(* Logix 5000 project; controller Receptivo vendor 1 type 14 code 106 rev 30.11; software revision 30.00; part 5 of 10 *)
(* tags used below, declared in another part *)
   Codigo_QAD1_Espacios : DINT;
   Descripcion1_Espacios : DINT;
   Descripcion2_Espacios : DINT;
   Numero_Espacios_Descripcion_1 : DINT;
   Numero_Espacios_Descripcion_2 : DINT;
   Numero_Espacios_QAD1 : DINT;
   Numero_Espacios_QAD2 : DINT;
   Print1_Ejecute : BOOL;
   Print1_OK : BOOL;
   Print2_Ejecute : BOOL;
   Print2_OK : BOOL;
   CAJAS_1 : DINT;
   CAJAS_2 : DINT;
   Calendario : Hora_y_Fecha;
   Cant_total : SINT;
   CERO : DINT;
   Clima_1 : DINT;
   Clima_2 : DINT;
   Codigo_QAD2_Espacios : DINT;
   Consecutivo : INT;
   Consecutivo_String : Consecutivo;
   Consolidado_Est : UDT_COLA[50];
   Counter_R_Estacion1 : COUNTER;
   Counter_R_Estacion2 : COUNTER;
   Counter_R_Estacion3 : COUNTER;
   Counter_R_Estacion4 : COUNTER;
   Densidad_1 : REAL;
   Densidad_2 : REAL;
   Densidad_Elmar_1 : REAL;
   Densidad_Fogg1_1 : REAL;
   EAN14_1 : Codigo_Barras;
   EAN14_2 : Codigo_Barras;
   Espacios : STRING;
   ESTACION_1 : DINT;
   Estacion_1_GCola_1 : UDT_COLA;
   Estacion_1_General : UDT_GENERAL;
   Estacion_1_Resumen : UDT_COLA[20];
   Estacion_1_String : STRING;
   ESTACION_2 : DINT;
   Estacion_2_GCola_1 : UDT_COLA;
   Estacion_2_General : UDT_GENERAL;
   Estacion_2_Resumen : UDT_COLA[20];
   Estacion_2_String : STRING;
   Estacion_3_Resumen : UDT_COLA[20];
   Estacion_4_Resumen : UDT_COLA[20];
   Forx : SINT;
   Fory : SINT;
   Forz : SINT;
   found : SINT;
   LInea_General_1 : INT;
   LInea_General_2 : INT;
   Linea_String_General : STRING;
   Lote : DINT;
   Operador_1 : DINT;
   Operador_2 : DINT;
   Pesaje_1 : REAL;
   Pesaje_2 : REAL;
   Peso_Caja_Elmar_1 : REAL;
   Peso_Caja_Fogg1_1 : REAL;
   PESO_REAL_1 : DINT;
   PESO_REAL_2 : DINT;
   PESO_TEORICO_1 : DINT;
   PESO_TEORICO_2 : DINT;
   Producido_Elmar_Ahora : UDT_Maestro;
   Producido_Fogg1_Ahora : UDT_Maestro;
   Producto1 : UDT_Inventario;
   Producto2 : UDT_Inventario;
   QAD_1 : STRING;
   QAD_2 : STRING;
(* MainProgram, continued *)

ROUTINE Consecutivo   (* ladder *)
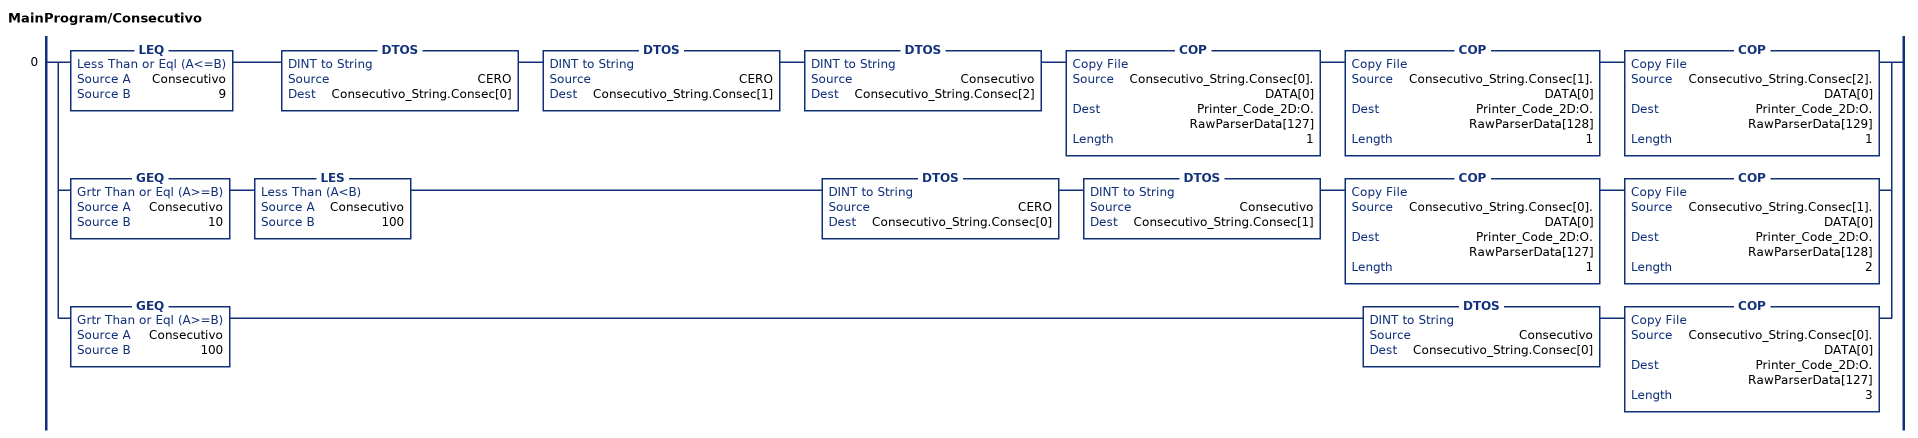
   0: [LEQ(Consecutivo,9) DTOS(CERO,Consecutivo_String.Consec[0]) DTOS(CERO,Consecutivo_String.Consec[1]) DTOS(Consecutivo,Consecutivo_String.Consec[2]) COP(Consecutivo_String.Consec[0].DATA[0],Printer_Code_2D:O.RawParserData[127],1) COP(Consecutivo_String.Consec[1].DATA[0],Printer_Code_2D:O.RawParserData[128],1) COP(Consecutivo_String.Consec[2].DATA[0],Printer_Code_2D:O.RawParserData[129],1) ,GEQ(Consecutivo,10) LES(Consecutivo,100) DTOS(CERO,Consecutivo_String.Consec[0]) DTOS(Consecutivo,Consecutivo_String.Consec[1]) COP(Consecutivo_String.Consec[0].DATA[0],Printer_Code_2D:O.RawParserData[127],1) COP(Consecutivo_String.Consec[1].DATA[0],Printer_Code_2D:O.RawParserData[128],2) ,GEQ(Consecutivo,100) DTOS(Consecutivo,Consecutivo_String.Consec[0]) COP(Consecutivo_String.Consec[0].DATA[0],Printer_Code_2D:O.RawParserData[127],3) ];
END_ROUTINE

ROUTINE Consolidado   (* ladder *)
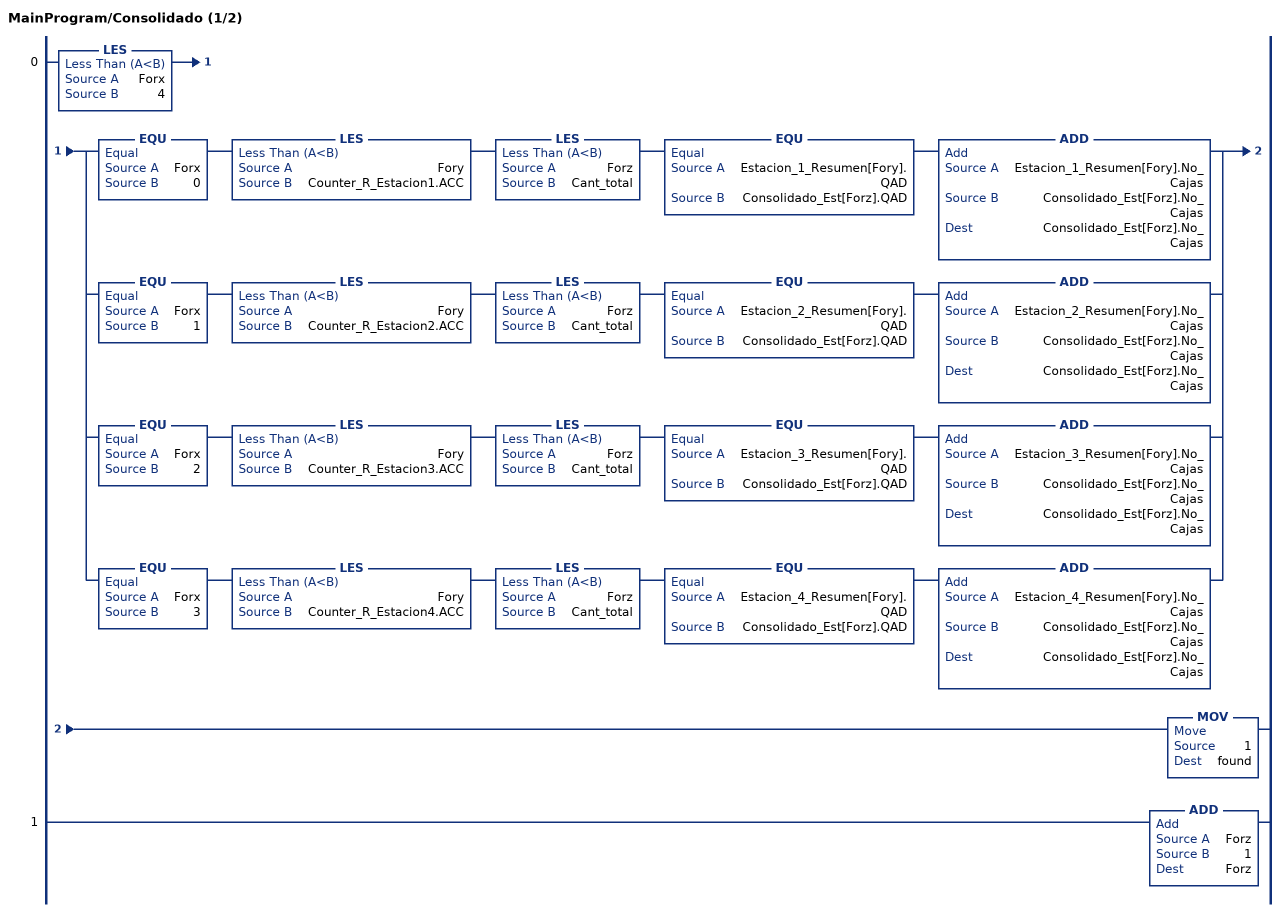
   0: LES(Forx,4)[EQU(Forx,0) LES(Fory,Counter_R_Estacion1.ACC) LES(Forz,Cant_total) EQU(Estacion_1_Resumen[Fory].QAD,Consolidado_Est[Forz].QAD) ADD(Estacion_1_Resumen[Fory].No_Cajas,Consolidado_Est[Forz].No_Cajas,Consolidado_Est[Forz].No_Cajas) ,EQU(Forx,1) LES(Fory,Counter_R_Estacion2.ACC) LES(Forz,Cant_total) EQU(Estacion_2_Resumen[Fory].QAD,Consolidado_Est[Forz].QAD) ADD(Estacion_2_Resumen[Fory].No_Cajas,Consolidado_Est[Forz].No_Cajas,Consolidado_Est[Forz].No_Cajas) ,EQU(Forx,2) LES(Fory,Counter_R_Estacion3.ACC) LES(Forz,Cant_total) EQU(Estacion_3_Resumen[Fory].QAD,Consolidado_Est[Forz].QAD) ADD(Estacion_3_Resumen[Fory].No_Cajas,Consolidado_Est[Forz].No_Cajas,Consolidado_Est[Forz].No_Cajas) ,EQU(Forx,3) LES(Fory,Counter_R_Estacion4.ACC) LES(Forz,Cant_total) EQU(Estacion_4_Resumen[Fory].QAD,Consolidado_Est[Forz].QAD) ADD(Estacion_4_Resumen[Fory].No_Cajas,Consolidado_Est[Forz].No_Cajas,Consolidado_Est[Forz].No_Cajas) ]MOV(1,found);
   1: ADD(Forz,1,Forz);
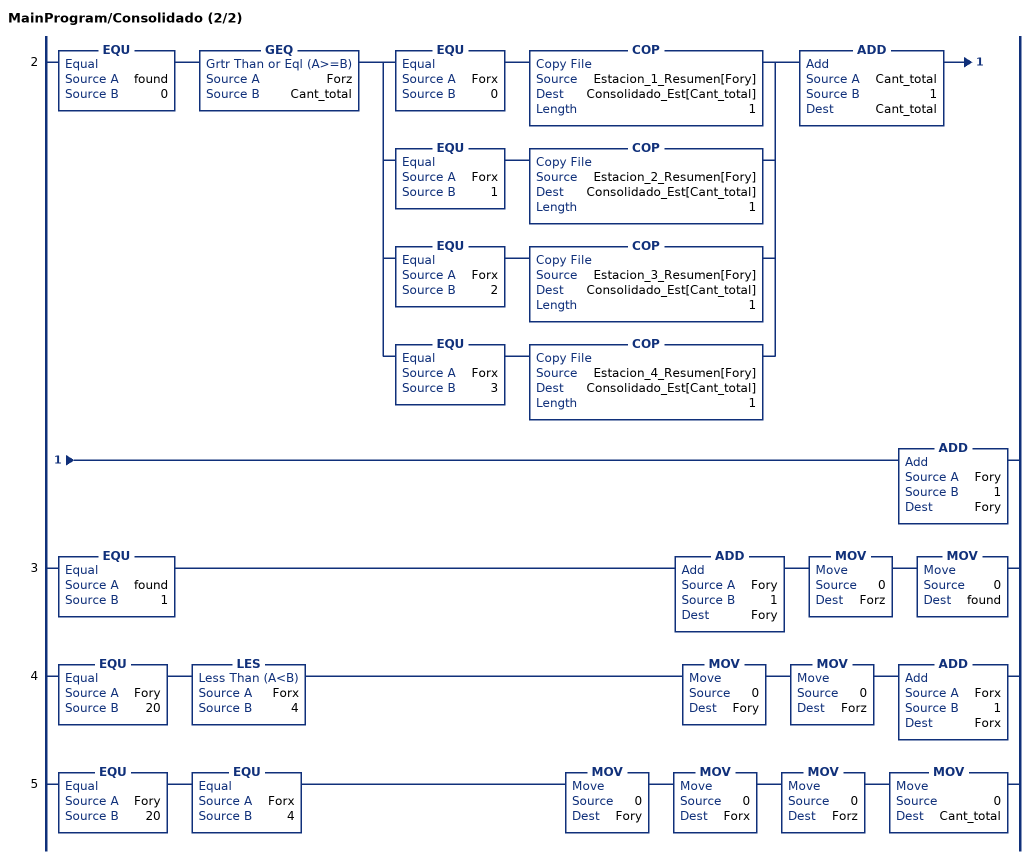
   2: EQU(found,0)GEQ(Forz,Cant_total)[EQU(Forx,0) COP(Estacion_1_Resumen[Fory],Consolidado_Est[Cant_total],1) ,EQU(Forx,1) COP(Estacion_2_Resumen[Fory],Consolidado_Est[Cant_total],1) ,EQU(Forx,2) COP(Estacion_3_Resumen[Fory],Consolidado_Est[Cant_total],1) ,EQU(Forx,3) COP(Estacion_4_Resumen[Fory],Consolidado_Est[Cant_total],1) ]ADD(Cant_total,1,Cant_total)ADD(Fory,1,Fory);
   3: EQU(found,1)ADD(Fory,1,Fory)MOV(0,Forz)MOV(0,found);
   4: EQU(Fory,20)LES(Forx,4)MOV(0,Fory)MOV(0,Forz)ADD(Forx,1,Forx);
   5: EQU(Fory,20)EQU(Forx,4)MOV(0,Fory)MOV(0,Forx)MOV(0,Forz)MOV(0,Cant_total);
END_ROUTINE

ROUTINE Copy_To_Parser_Standard   (* ladder *)
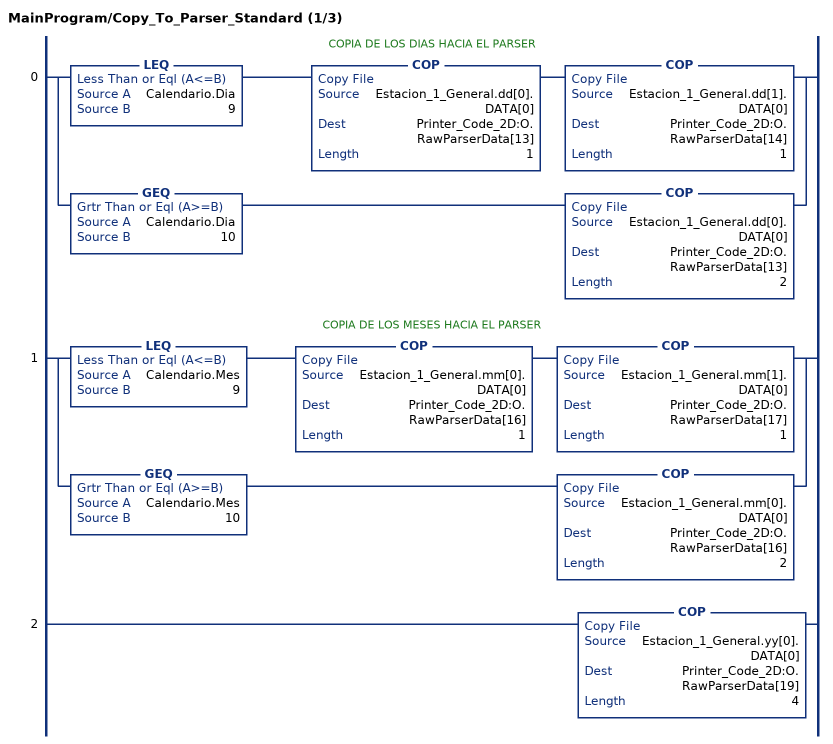
   // COPIA DE LOS DIAS HACIA EL PARSER
   0: [LEQ(Calendario.Dia,9) COP(Estacion_1_General.dd[0].DATA[0],Printer_Code_2D:O.RawParserData[13],1) COP(Estacion_1_General.dd[1].DATA[0],Printer_Code_2D:O.RawParserData[14],1) ,GEQ(Calendario.Dia,10) COP(Estacion_1_General.dd[0].DATA[0],Printer_Code_2D:O.RawParserData[13],2) ];
   // COPIA DE LOS MESES HACIA EL PARSER
   1: [LEQ(Calendario.Mes,9) COP(Estacion_1_General.mm[0].DATA[0],Printer_Code_2D:O.RawParserData[16],1) COP(Estacion_1_General.mm[1].DATA[0],Printer_Code_2D:O.RawParserData[17],1) ,GEQ(Calendario.Mes,10) COP(Estacion_1_General.mm[0].DATA[0],Printer_Code_2D:O.RawParserData[16],2) ];
   2: COP(Estacion_1_General.yy[0].DATA[0],Printer_Code_2D:O.RawParserData[19],4);
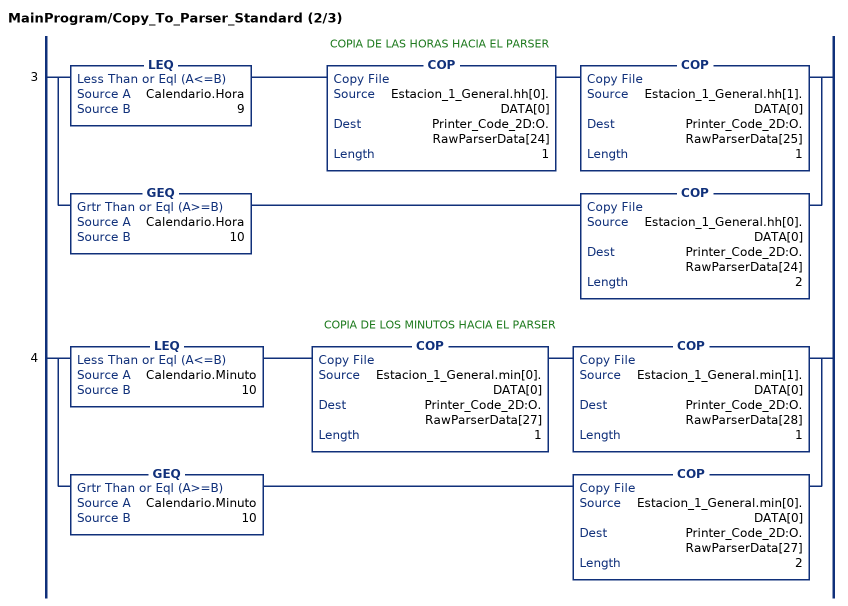
   // COPIA DE LAS HORAS HACIA EL PARSER
   3: [LEQ(Calendario.Hora,9) COP(Estacion_1_General.hh[0].DATA[0],Printer_Code_2D:O.RawParserData[24],1) COP(Estacion_1_General.hh[1].DATA[0],Printer_Code_2D:O.RawParserData[25],1) ,GEQ(Calendario.Hora,10) COP(Estacion_1_General.hh[0].DATA[0],Printer_Code_2D:O.RawParserData[24],2) ];
   // COPIA DE LOS MINUTOS HACIA EL PARSER
   4: [LEQ(Calendario.Minuto,10) COP(Estacion_1_General.min[0].DATA[0],Printer_Code_2D:O.RawParserData[27],1) COP(Estacion_1_General.min[1].DATA[0],Printer_Code_2D:O.RawParserData[28],1) ,GEQ(Calendario.Minuto,10) COP(Estacion_1_General.min[0].DATA[0],Printer_Code_2D:O.RawParserData[27],2) ];
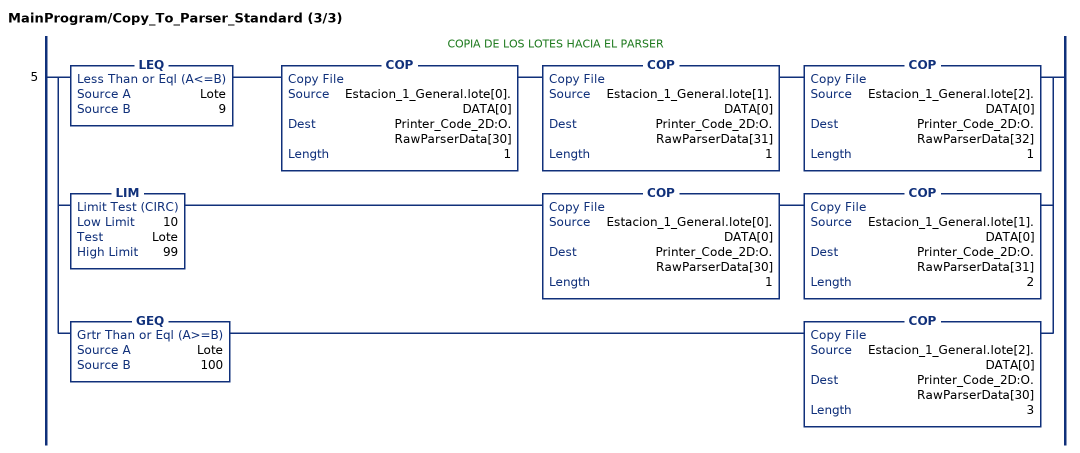
   // COPIA DE LOS LOTES HACIA EL PARSER
   5: [LEQ(Lote,9) COP(Estacion_1_General.lote[0].DATA[0],Printer_Code_2D:O.RawParserData[30],1) COP(Estacion_1_General.lote[1].DATA[0],Printer_Code_2D:O.RawParserData[31],1) COP(Estacion_1_General.lote[2].DATA[0],Printer_Code_2D:O.RawParserData[32],1) ,LIM(10,Lote,99) COP(Estacion_1_General.lote[0].DATA[0],Printer_Code_2D:O.RawParserData[30],1) COP(Estacion_1_General.lote[1].DATA[0],Printer_Code_2D:O.RawParserData[31],2) ,GEQ(Lote,100) COP(Estacion_1_General.lote[2].DATA[0],Printer_Code_2D:O.RawParserData[30],3) ];
END_ROUTINE

ROUTINE Estacion_1_Datos   (* ladder *)
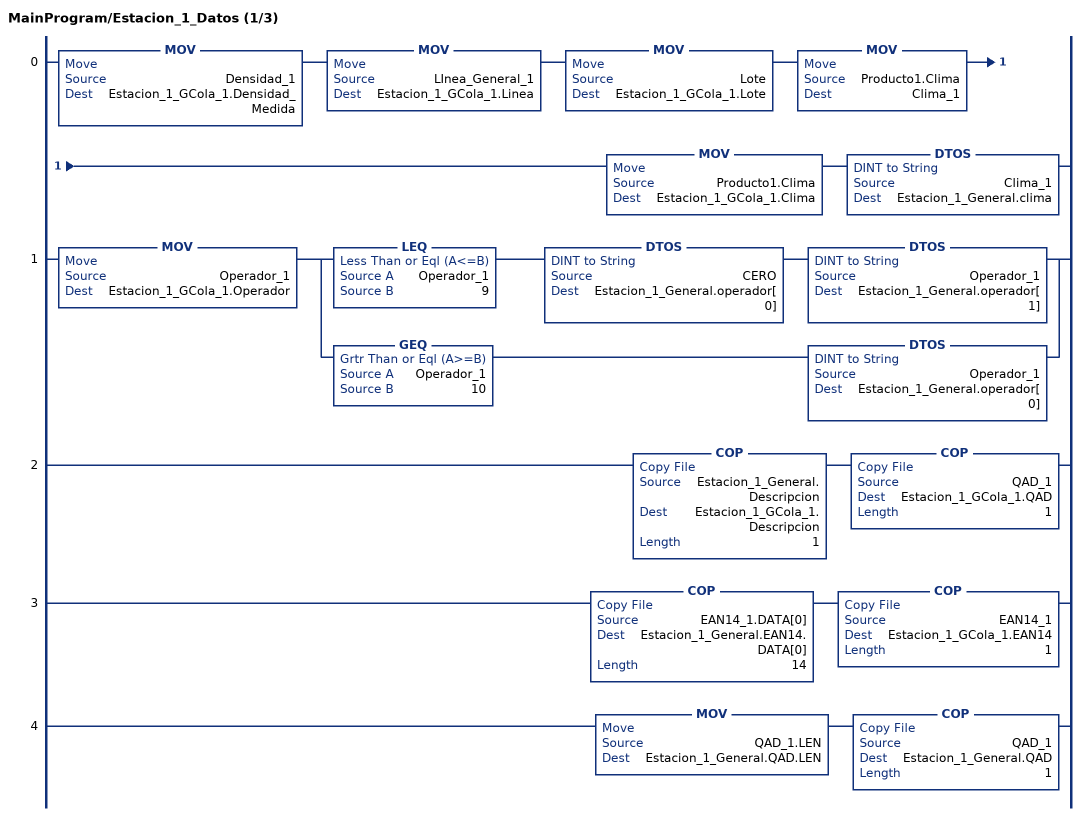
   0: MOV(Densidad_1,Estacion_1_GCola_1.Densidad_Medida)MOV(LInea_General_1,Estacion_1_GCola_1.Linea)MOV(Lote,Estacion_1_GCola_1.Lote)MOV(Producto1.Clima,Clima_1)MOV(Producto1.Clima,Estacion_1_GCola_1.Clima)DTOS(Clima_1,Estacion_1_General.clima);
   1: MOV(Operador_1,Estacion_1_GCola_1.Operador)[LEQ(Operador_1,9) DTOS(CERO,Estacion_1_General.operador[0]) DTOS(Operador_1,Estacion_1_General.operador[1]) ,GEQ(Operador_1,10) DTOS(Operador_1,Estacion_1_General.operador[0]) ];
   2: COP(Estacion_1_General.Descripcion,Estacion_1_GCola_1.Descripcion,1)COP(QAD_1,Estacion_1_GCola_1.QAD,1);
   3: COP(EAN14_1.DATA[0],Estacion_1_General.EAN14.DATA[0],14)COP(EAN14_1,Estacion_1_GCola_1.EAN14,1);
   4: MOV(QAD_1.LEN,Estacion_1_General.QAD.LEN)COP(QAD_1,Estacion_1_General.QAD,1);
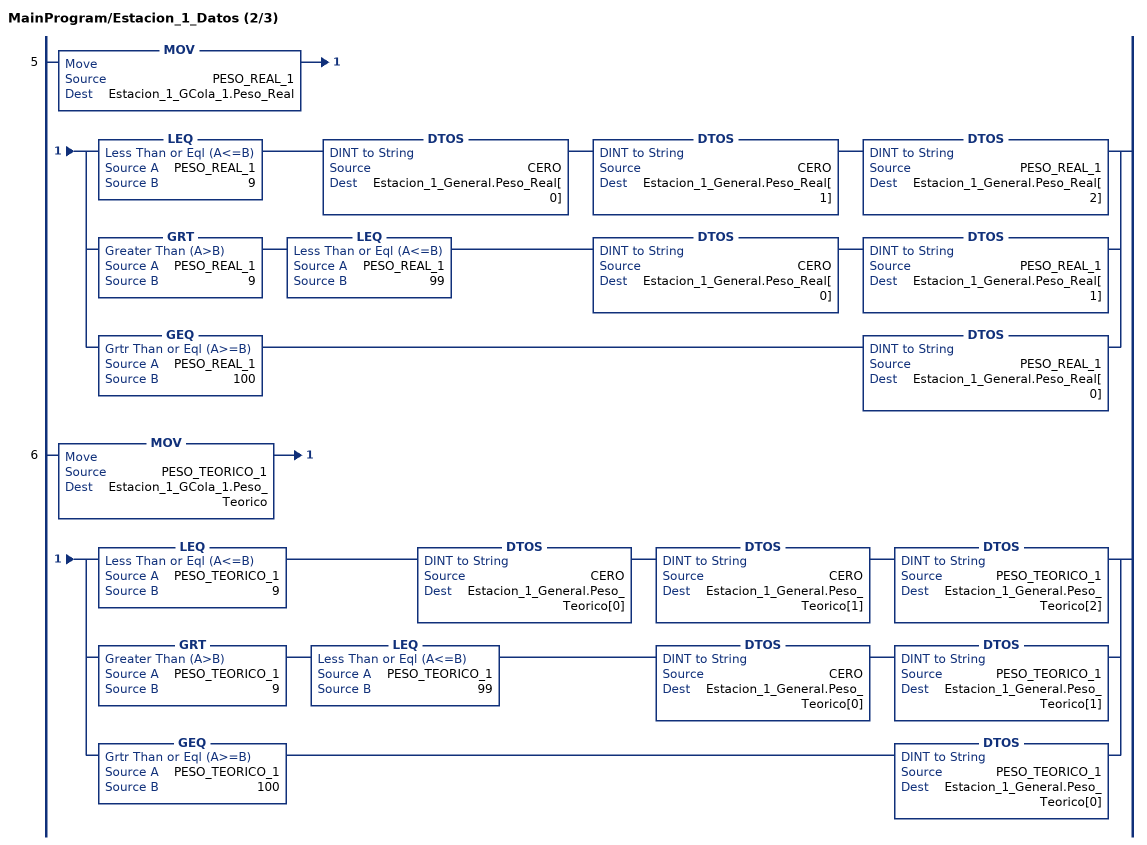
   5: MOV(PESO_REAL_1,Estacion_1_GCola_1.Peso_Real)[LEQ(PESO_REAL_1,9) DTOS(CERO,Estacion_1_General.Peso_Real[0]) DTOS(CERO,Estacion_1_General.Peso_Real[1]) DTOS(PESO_REAL_1,Estacion_1_General.Peso_Real[2]) ,GRT(PESO_REAL_1,9) LEQ(PESO_REAL_1,99) DTOS(CERO,Estacion_1_General.Peso_Real[0]) DTOS(PESO_REAL_1,Estacion_1_General.Peso_Real[1]) ,GEQ(PESO_REAL_1,100) DTOS(PESO_REAL_1,Estacion_1_General.Peso_Real[0]) ];
   6: MOV(PESO_TEORICO_1,Estacion_1_GCola_1.Peso_Teorico)[LEQ(PESO_TEORICO_1,9) DTOS(CERO,Estacion_1_General.Peso_Teorico[0]) DTOS(CERO,Estacion_1_General.Peso_Teorico[1]) DTOS(PESO_TEORICO_1,Estacion_1_General.Peso_Teorico[2]) ,GRT(PESO_TEORICO_1,9) LEQ(PESO_TEORICO_1,99) DTOS(CERO,Estacion_1_General.Peso_Teorico[0]) DTOS(PESO_TEORICO_1,Estacion_1_General.Peso_Teorico[1]) ,GEQ(PESO_TEORICO_1,100) DTOS(PESO_TEORICO_1,Estacion_1_General.Peso_Teorico[0]) ];
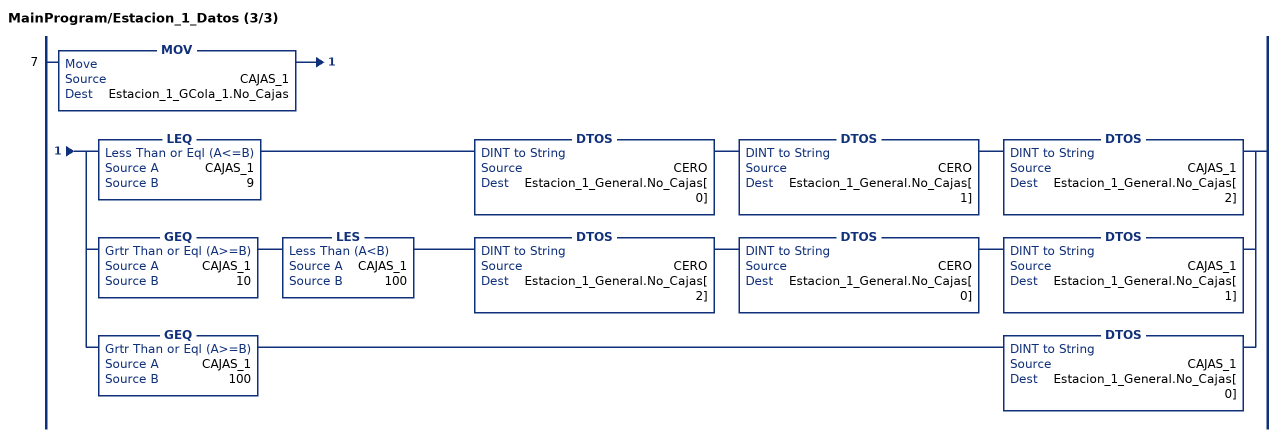
   7: MOV(CAJAS_1,Estacion_1_GCola_1.No_Cajas)[LEQ(CAJAS_1,9) DTOS(CERO,Estacion_1_General.No_Cajas[0]) DTOS(CERO,Estacion_1_General.No_Cajas[1]) DTOS(CAJAS_1,Estacion_1_General.No_Cajas[2]) ,GEQ(CAJAS_1,10) LES(CAJAS_1,100) DTOS(CERO,Estacion_1_General.No_Cajas[2]) DTOS(CERO,Estacion_1_General.No_Cajas[0]) DTOS(CAJAS_1,Estacion_1_General.No_Cajas[1]) ,GEQ(CAJAS_1,100) DTOS(CAJAS_1,Estacion_1_General.No_Cajas[0]) ];
END_ROUTINE

ROUTINE Estacion_1_To_Printer   (* ladder *)
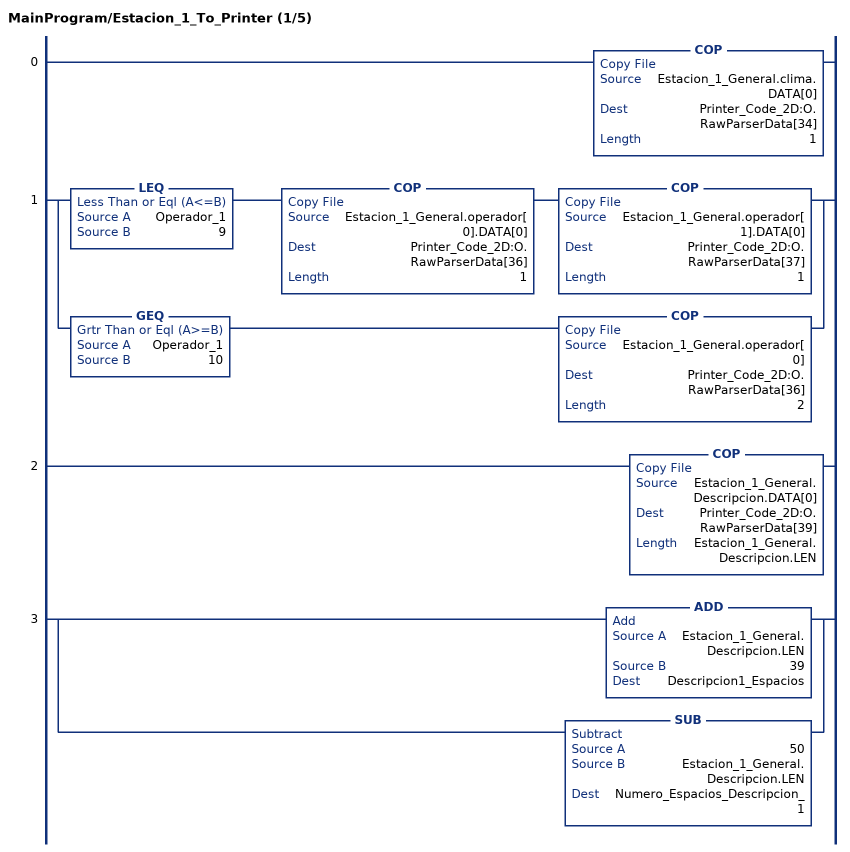
   0: COP(Estacion_1_General.clima.DATA[0],Printer_Code_2D:O.RawParserData[34],1);
   1: [LEQ(Operador_1,9) COP(Estacion_1_General.operador[0].DATA[0],Printer_Code_2D:O.RawParserData[36],1) COP(Estacion_1_General.operador[1].DATA[0],Printer_Code_2D:O.RawParserData[37],1) ,GEQ(Operador_1,10) COP(Estacion_1_General.operador[0],Printer_Code_2D:O.RawParserData[36],2) ];
   2: COP(Estacion_1_General.Descripcion.DATA[0],Printer_Code_2D:O.RawParserData[39],Estacion_1_General.Descripcion.LEN);
   3: [ADD(Estacion_1_General.Descripcion.LEN,39,Descripcion1_Espacios) ,SUB(50,Estacion_1_General.Descripcion.LEN,Numero_Espacios_Descripcion_1) ];
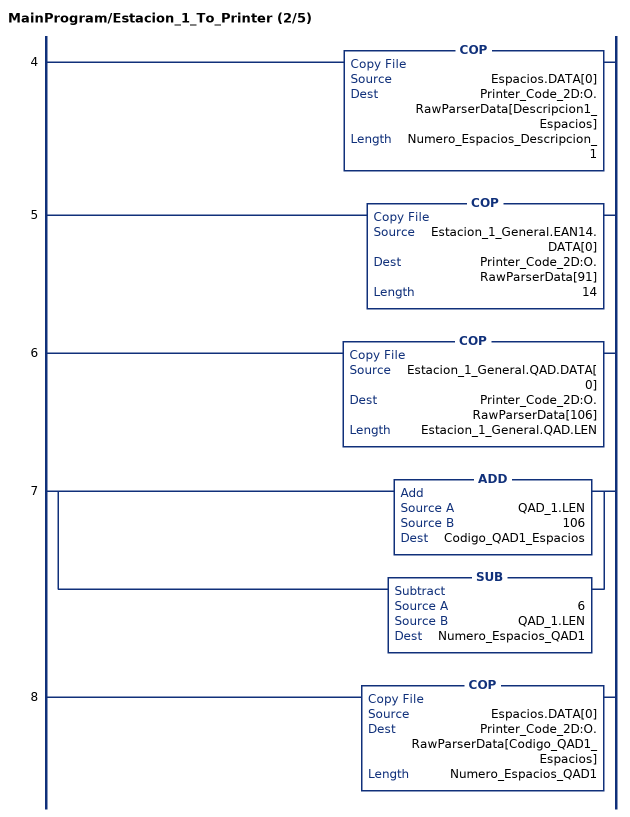
   4: COP(Espacios.DATA[0],Printer_Code_2D:O.RawParserData[Descripcion1_Espacios],Numero_Espacios_Descripcion_1);
   5: COP(Estacion_1_General.EAN14.DATA[0],Printer_Code_2D:O.RawParserData[91],14);
   6: COP(Estacion_1_General.QAD.DATA[0],Printer_Code_2D:O.RawParserData[106],Estacion_1_General.QAD.LEN);
   7: [ADD(QAD_1.LEN,106,Codigo_QAD1_Espacios) ,SUB(6,QAD_1.LEN,Numero_Espacios_QAD1) ];
   8: COP(Espacios.DATA[0],Printer_Code_2D:O.RawParserData[Codigo_QAD1_Espacios],Numero_Espacios_QAD1);
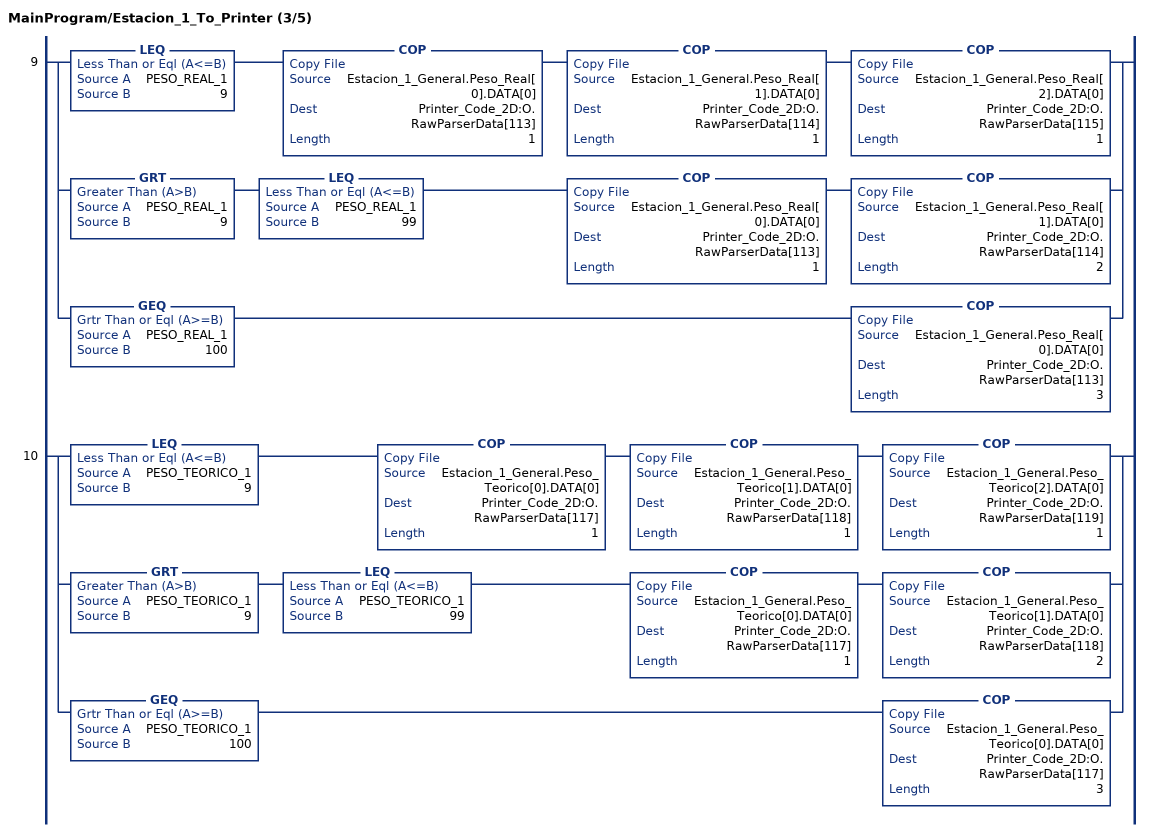
   9: [LEQ(PESO_REAL_1,9) COP(Estacion_1_General.Peso_Real[0].DATA[0],Printer_Code_2D:O.RawParserData[113],1) COP(Estacion_1_General.Peso_Real[1].DATA[0],Printer_Code_2D:O.RawParserData[114],1) COP(Estacion_1_General.Peso_Real[2].DATA[0],Printer_Code_2D:O.RawParserData[115],1) ,GRT(PESO_REAL_1,9) LEQ(PESO_REAL_1,99) COP(Estacion_1_General.Peso_Real[0].DATA[0],Printer_Code_2D:O.RawParserData[113],1) COP(Estacion_1_General.Peso_Real[1].DATA[0],Printer_Code_2D:O.RawParserData[114],2) ,GEQ(PESO_REAL_1,100) COP(Estacion_1_General.Peso_Real[0].DATA[0],Printer_Code_2D:O.RawParserData[113],3) ];
   10: [LEQ(PESO_TEORICO_1,9) COP(Estacion_1_General.Peso_Teorico[0].DATA[0],Printer_Code_2D:O.RawParserData[117],1) COP(Estacion_1_General.Peso_Teorico[1].DATA[0],Printer_Code_2D:O.RawParserData[118],1) COP(Estacion_1_General.Peso_Teorico[2].DATA[0],Printer_Code_2D:O.RawParserData[119],1) ,GRT(PESO_TEORICO_1,9) LEQ(PESO_TEORICO_1,99) COP(Estacion_1_General.Peso_Teorico[0].DATA[0],Printer_Code_2D:O.RawParserData[117],1) COP(Estacion_1_General.Peso_Teorico[1].DATA[0],Printer_Code_2D:O.RawParserData[118],2) ,GEQ(PESO_TEORICO_1,100) COP(Estacion_1_General.Peso_Teorico[0].DATA[0],Printer_Code_2D:O.RawParserData[117],3) ];
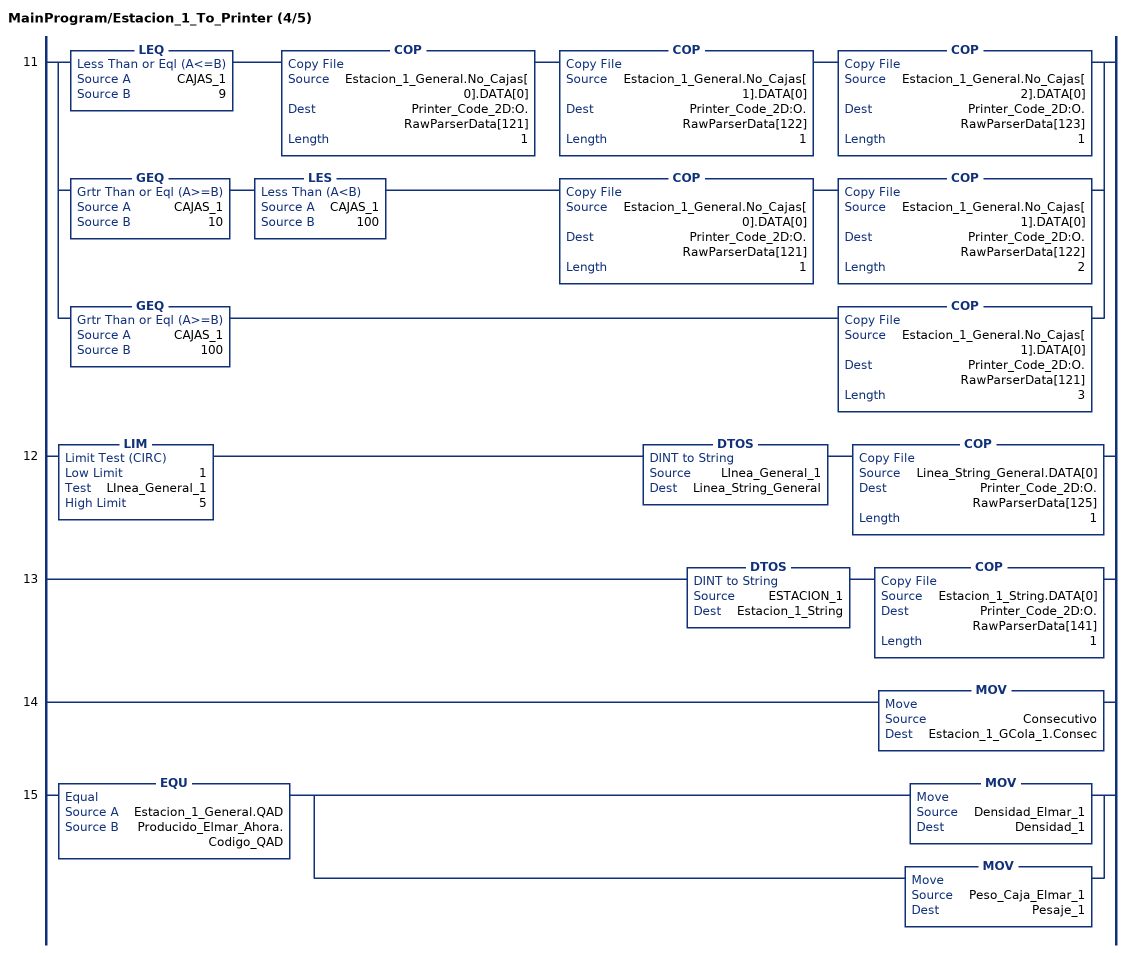
   11: [LEQ(CAJAS_1,9) COP(Estacion_1_General.No_Cajas[0].DATA[0],Printer_Code_2D:O.RawParserData[121],1) COP(Estacion_1_General.No_Cajas[1].DATA[0],Printer_Code_2D:O.RawParserData[122],1) COP(Estacion_1_General.No_Cajas[2].DATA[0],Printer_Code_2D:O.RawParserData[123],1) ,GEQ(CAJAS_1,10) LES(CAJAS_1,100) COP(Estacion_1_General.No_Cajas[0].DATA[0],Printer_Code_2D:O.RawParserData[121],1) COP(Estacion_1_General.No_Cajas[1].DATA[0],Printer_Code_2D:O.RawParserData[122],2) ,GEQ(CAJAS_1,100) COP(Estacion_1_General.No_Cajas[1].DATA[0],Printer_Code_2D:O.RawParserData[121],3) ];
   12: LIM(1,LInea_General_1,5)DTOS(LInea_General_1,Linea_String_General)COP(Linea_String_General.DATA[0],Printer_Code_2D:O.RawParserData[125],1);
   13: DTOS(ESTACION_1,Estacion_1_String)COP(Estacion_1_String.DATA[0],Printer_Code_2D:O.RawParserData[141],1);
   14: MOV(Consecutivo,Estacion_1_GCola_1.Consec);
   15: EQU(Estacion_1_General.QAD,Producido_Elmar_Ahora.Codigo_QAD)[MOV(Densidad_Elmar_1,Densidad_1) ,MOV(Peso_Caja_Elmar_1,Pesaje_1) ];
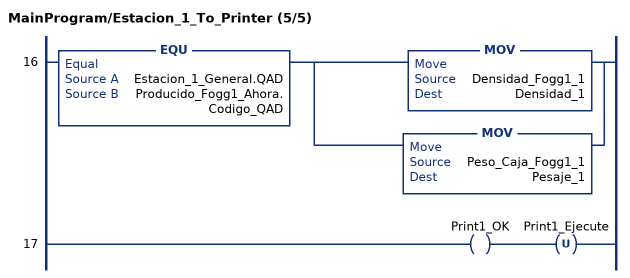
   16: EQU(Estacion_1_General.QAD,Producido_Fogg1_Ahora.Codigo_QAD)[MOV(Densidad_Fogg1_1,Densidad_1) ,MOV(Peso_Caja_Fogg1_1,Pesaje_1) ];
   17: OTE(Print1_OK)OTU(Print1_Ejecute);
END_ROUTINE

ROUTINE Estacion_2_Datos   (* ladder *)
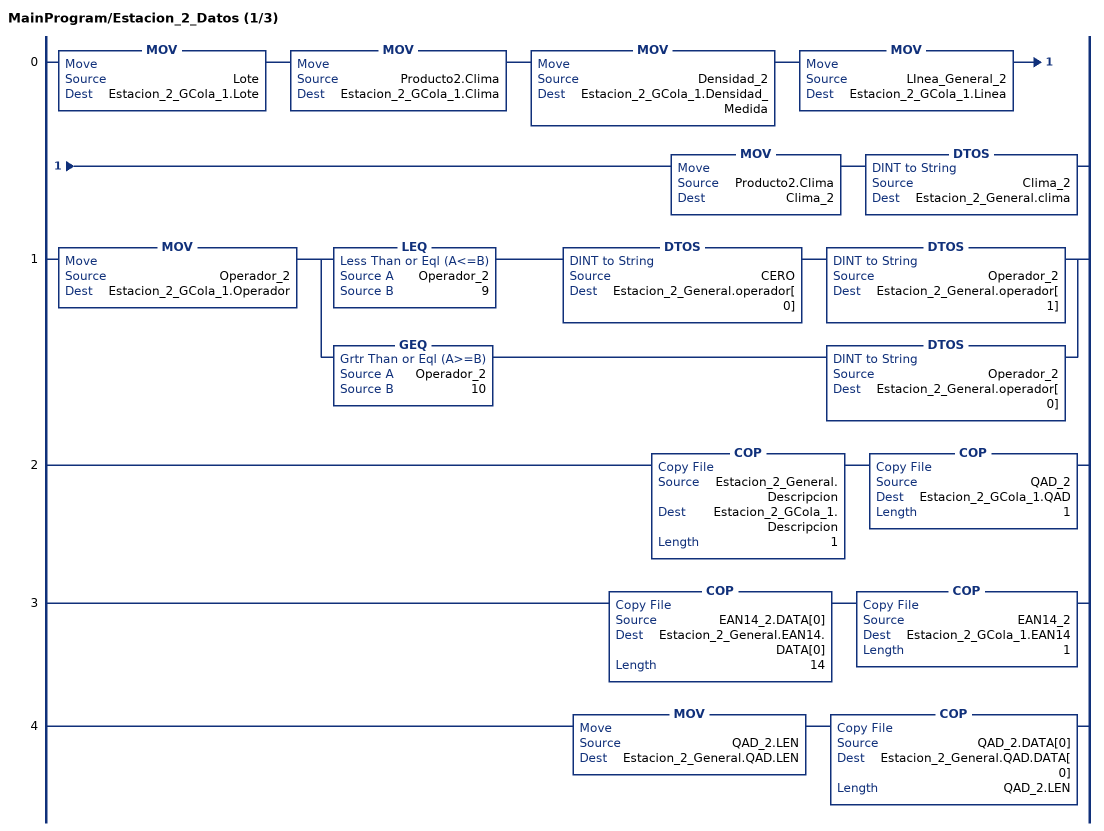
   0: MOV(Lote,Estacion_2_GCola_1.Lote)MOV(Producto2.Clima,Estacion_2_GCola_1.Clima)MOV(Densidad_2,Estacion_2_GCola_1.Densidad_Medida)MOV(LInea_General_2,Estacion_2_GCola_1.Linea)MOV(Producto2.Clima,Clima_2)DTOS(Clima_2,Estacion_2_General.clima);
   1: MOV(Operador_2,Estacion_2_GCola_1.Operador)[LEQ(Operador_2,9) DTOS(CERO,Estacion_2_General.operador[0]) DTOS(Operador_2,Estacion_2_General.operador[1]) ,GEQ(Operador_2,10) DTOS(Operador_2,Estacion_2_General.operador[0]) ];
   2: COP(Estacion_2_General.Descripcion,Estacion_2_GCola_1.Descripcion,1)COP(QAD_2,Estacion_2_GCola_1.QAD,1);
   3: COP(EAN14_2.DATA[0],Estacion_2_General.EAN14.DATA[0],14)COP(EAN14_2,Estacion_2_GCola_1.EAN14,1);
   4: MOV(QAD_2.LEN,Estacion_2_General.QAD.LEN)COP(QAD_2.DATA[0],Estacion_2_General.QAD.DATA[0],QAD_2.LEN);
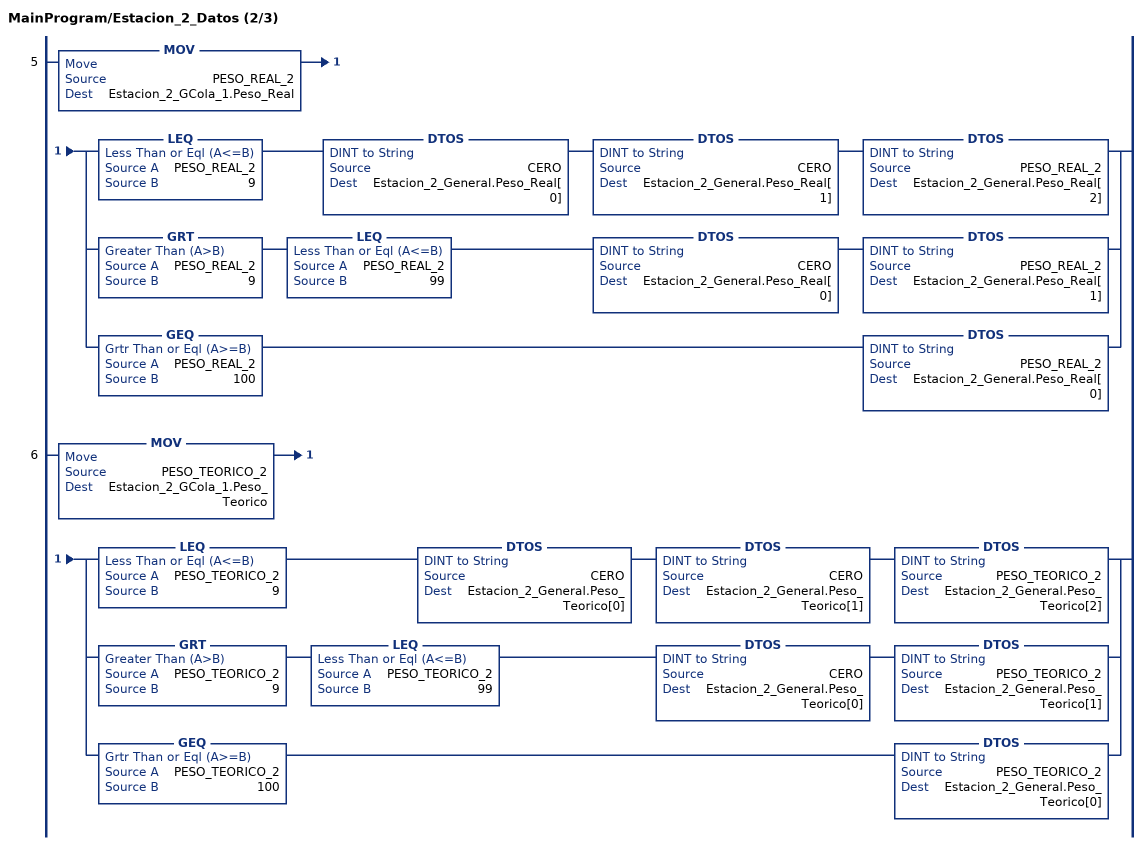
   5: MOV(PESO_REAL_2,Estacion_2_GCola_1.Peso_Real)[LEQ(PESO_REAL_2,9) DTOS(CERO,Estacion_2_General.Peso_Real[0]) DTOS(CERO,Estacion_2_General.Peso_Real[1]) DTOS(PESO_REAL_2,Estacion_2_General.Peso_Real[2]) ,GRT(PESO_REAL_2,9) LEQ(PESO_REAL_2,99) DTOS(CERO,Estacion_2_General.Peso_Real[0]) DTOS(PESO_REAL_2,Estacion_2_General.Peso_Real[1]) ,GEQ(PESO_REAL_2,100) DTOS(PESO_REAL_2,Estacion_2_General.Peso_Real[0]) ];
   6: MOV(PESO_TEORICO_2,Estacion_2_GCola_1.Peso_Teorico)[LEQ(PESO_TEORICO_2,9) DTOS(CERO,Estacion_2_General.Peso_Teorico[0]) DTOS(CERO,Estacion_2_General.Peso_Teorico[1]) DTOS(PESO_TEORICO_2,Estacion_2_General.Peso_Teorico[2]) ,GRT(PESO_TEORICO_2,9) LEQ(PESO_TEORICO_2,99) DTOS(CERO,Estacion_2_General.Peso_Teorico[0]) DTOS(PESO_TEORICO_2,Estacion_2_General.Peso_Teorico[1]) ,GEQ(PESO_TEORICO_2,100) DTOS(PESO_TEORICO_2,Estacion_2_General.Peso_Teorico[0]) ];
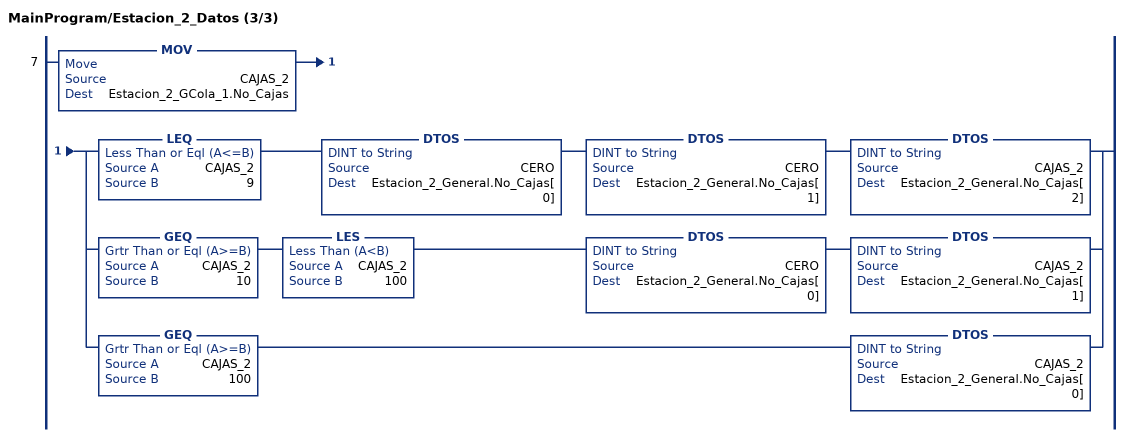
   7: MOV(CAJAS_2,Estacion_2_GCola_1.No_Cajas)[LEQ(CAJAS_2,9) DTOS(CERO,Estacion_2_General.No_Cajas[0]) DTOS(CERO,Estacion_2_General.No_Cajas[1]) DTOS(CAJAS_2,Estacion_2_General.No_Cajas[2]) ,GEQ(CAJAS_2,10) LES(CAJAS_2,100) DTOS(CERO,Estacion_2_General.No_Cajas[0]) DTOS(CAJAS_2,Estacion_2_General.No_Cajas[1]) ,GEQ(CAJAS_2,100) DTOS(CAJAS_2,Estacion_2_General.No_Cajas[0]) ];
END_ROUTINE

ROUTINE Estacion_2_To_Printer   (* ladder *)
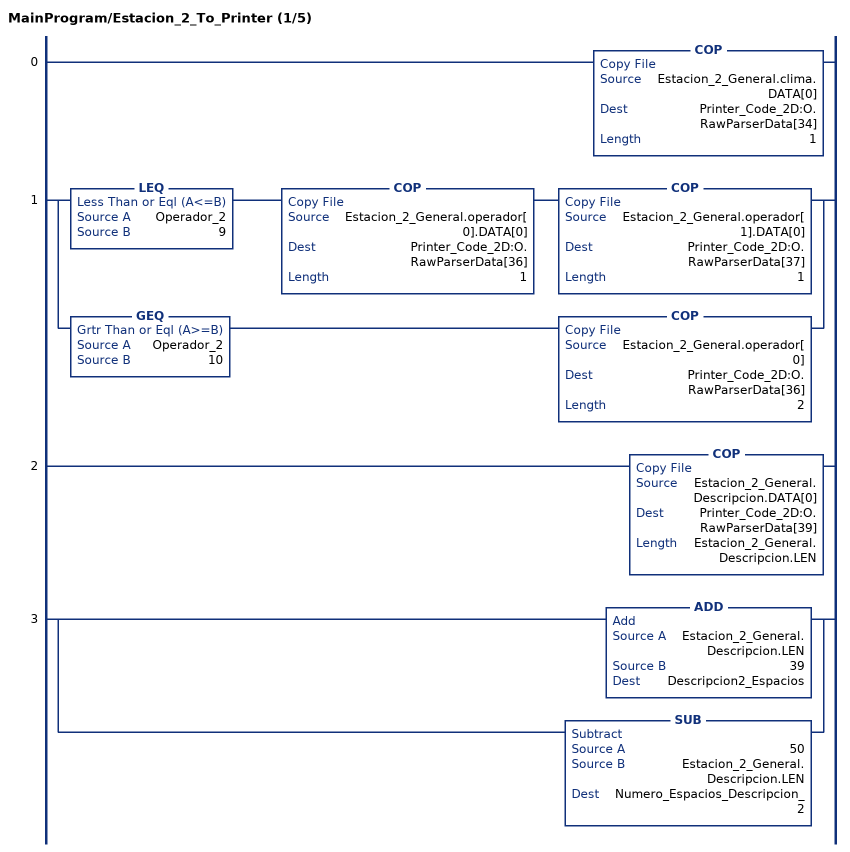
   0: COP(Estacion_2_General.clima.DATA[0],Printer_Code_2D:O.RawParserData[34],1);
   1: [LEQ(Operador_2,9) COP(Estacion_2_General.operador[0].DATA[0],Printer_Code_2D:O.RawParserData[36],1) COP(Estacion_2_General.operador[1].DATA[0],Printer_Code_2D:O.RawParserData[37],1) ,GEQ(Operador_2,10) COP(Estacion_2_General.operador[0],Printer_Code_2D:O.RawParserData[36],2) ];
   2: COP(Estacion_2_General.Descripcion.DATA[0],Printer_Code_2D:O.RawParserData[39],Estacion_2_General.Descripcion.LEN);
   3: [ADD(Estacion_2_General.Descripcion.LEN,39,Descripcion2_Espacios) ,SUB(50,Estacion_2_General.Descripcion.LEN,Numero_Espacios_Descripcion_2) ];
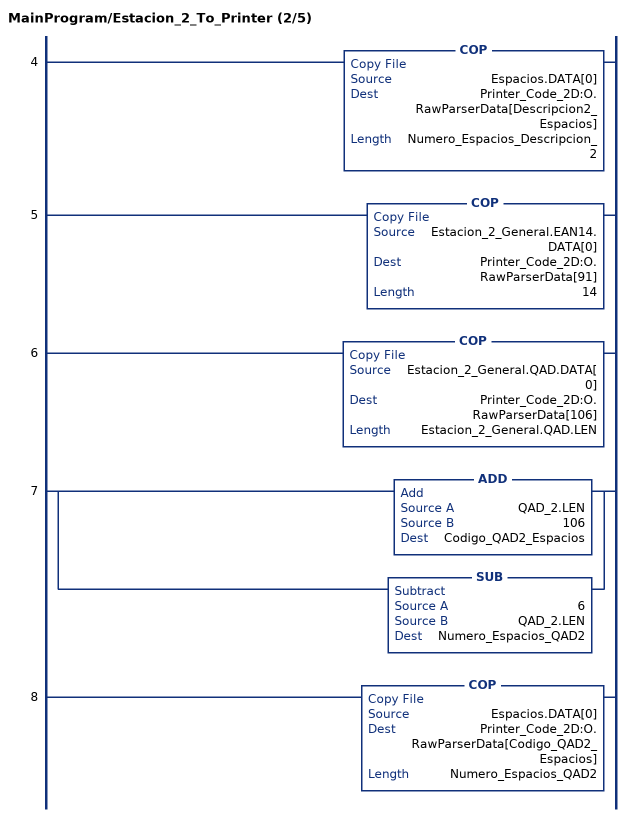
   4: COP(Espacios.DATA[0],Printer_Code_2D:O.RawParserData[Descripcion2_Espacios],Numero_Espacios_Descripcion_2);
   5: COP(Estacion_2_General.EAN14.DATA[0],Printer_Code_2D:O.RawParserData[91],14);
   6: COP(Estacion_2_General.QAD.DATA[0],Printer_Code_2D:O.RawParserData[106],Estacion_2_General.QAD.LEN);
   7: [ADD(QAD_2.LEN,106,Codigo_QAD2_Espacios) ,SUB(6,QAD_2.LEN,Numero_Espacios_QAD2) ];
   8: COP(Espacios.DATA[0],Printer_Code_2D:O.RawParserData[Codigo_QAD2_Espacios],Numero_Espacios_QAD2);
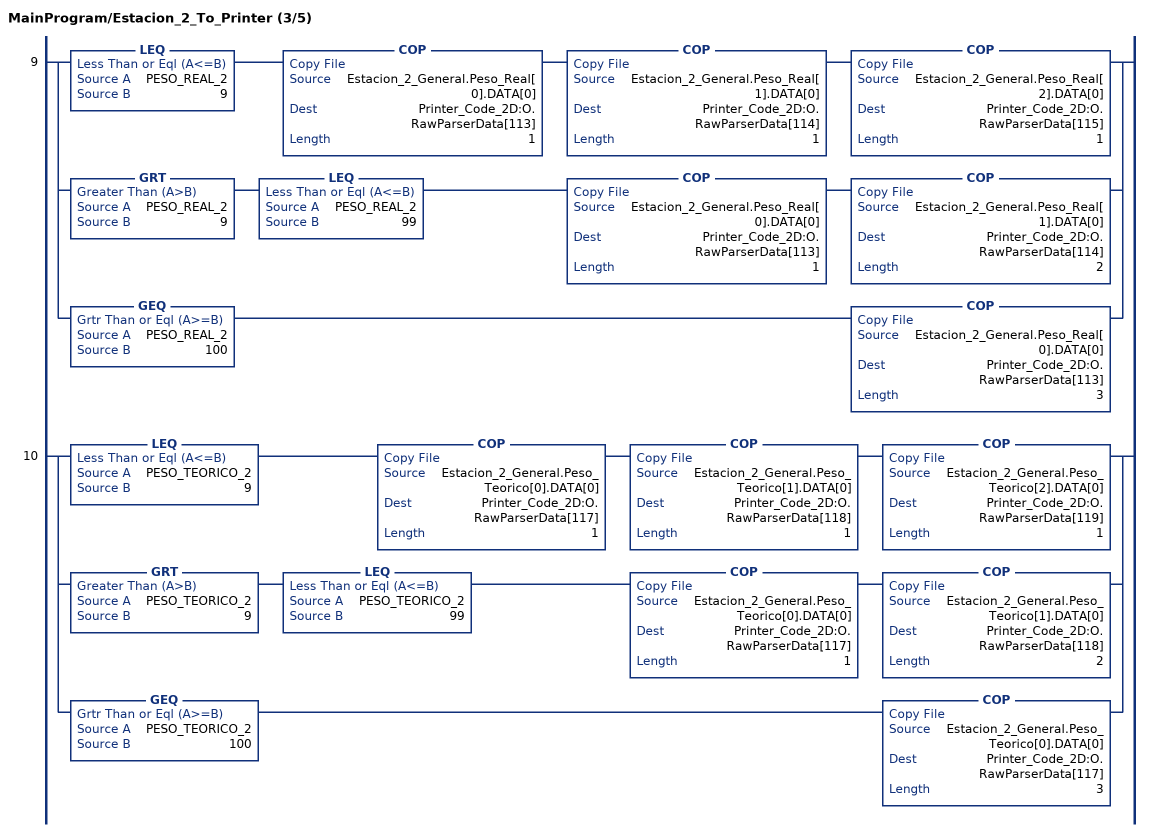
   9: [LEQ(PESO_REAL_2,9) COP(Estacion_2_General.Peso_Real[0].DATA[0],Printer_Code_2D:O.RawParserData[113],1) COP(Estacion_2_General.Peso_Real[1].DATA[0],Printer_Code_2D:O.RawParserData[114],1) COP(Estacion_2_General.Peso_Real[2].DATA[0],Printer_Code_2D:O.RawParserData[115],1) ,GRT(PESO_REAL_2,9) LEQ(PESO_REAL_2,99) COP(Estacion_2_General.Peso_Real[0].DATA[0],Printer_Code_2D:O.RawParserData[113],1) COP(Estacion_2_General.Peso_Real[1].DATA[0],Printer_Code_2D:O.RawParserData[114],2) ,GEQ(PESO_REAL_2,100) COP(Estacion_2_General.Peso_Real[0].DATA[0],Printer_Code_2D:O.RawParserData[113],3) ];
   10: [LEQ(PESO_TEORICO_2,9) COP(Estacion_2_General.Peso_Teorico[0].DATA[0],Printer_Code_2D:O.RawParserData[117],1) COP(Estacion_2_General.Peso_Teorico[1].DATA[0],Printer_Code_2D:O.RawParserData[118],1) COP(Estacion_2_General.Peso_Teorico[2].DATA[0],Printer_Code_2D:O.RawParserData[119],1) ,GRT(PESO_TEORICO_2,9) LEQ(PESO_TEORICO_2,99) COP(Estacion_2_General.Peso_Teorico[0].DATA[0],Printer_Code_2D:O.RawParserData[117],1) COP(Estacion_2_General.Peso_Teorico[1].DATA[0],Printer_Code_2D:O.RawParserData[118],2) ,GEQ(PESO_TEORICO_2,100) COP(Estacion_2_General.Peso_Teorico[0].DATA[0],Printer_Code_2D:O.RawParserData[117],3) ];
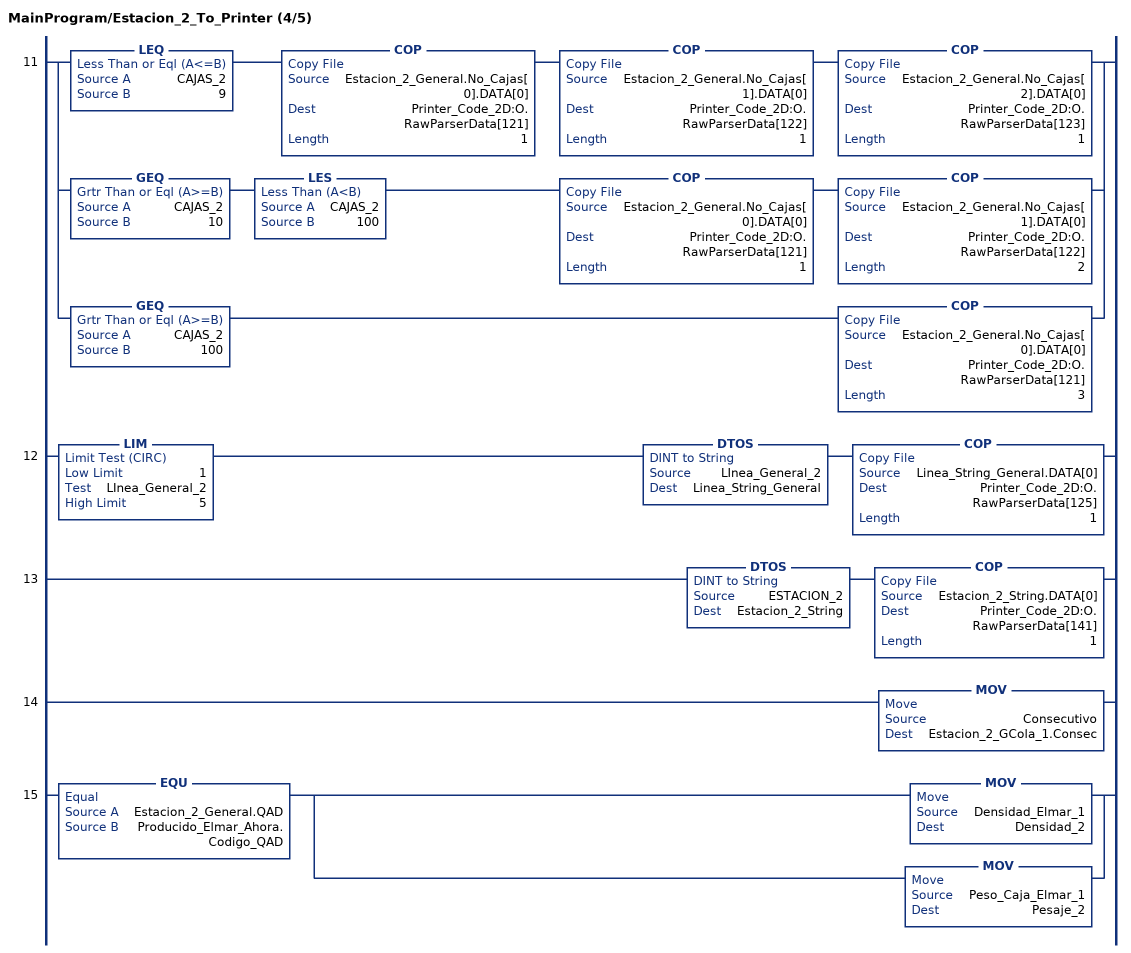
   11: [LEQ(CAJAS_2,9) COP(Estacion_2_General.No_Cajas[0].DATA[0],Printer_Code_2D:O.RawParserData[121],1) COP(Estacion_2_General.No_Cajas[1].DATA[0],Printer_Code_2D:O.RawParserData[122],1) COP(Estacion_2_General.No_Cajas[2].DATA[0],Printer_Code_2D:O.RawParserData[123],1) ,GEQ(CAJAS_2,10) LES(CAJAS_2,100) COP(Estacion_2_General.No_Cajas[0].DATA[0],Printer_Code_2D:O.RawParserData[121],1) COP(Estacion_2_General.No_Cajas[1].DATA[0],Printer_Code_2D:O.RawParserData[122],2) ,GEQ(CAJAS_2,100) COP(Estacion_2_General.No_Cajas[0].DATA[0],Printer_Code_2D:O.RawParserData[121],3) ];
   12: LIM(1,LInea_General_2,5)DTOS(LInea_General_2,Linea_String_General)COP(Linea_String_General.DATA[0],Printer_Code_2D:O.RawParserData[125],1);
   13: DTOS(ESTACION_2,Estacion_2_String)COP(Estacion_2_String.DATA[0],Printer_Code_2D:O.RawParserData[141],1);
   14: MOV(Consecutivo,Estacion_2_GCola_1.Consec);
   15: EQU(Estacion_2_General.QAD,Producido_Elmar_Ahora.Codigo_QAD)[MOV(Densidad_Elmar_1,Densidad_2) ,MOV(Peso_Caja_Elmar_1,Pesaje_2) ];
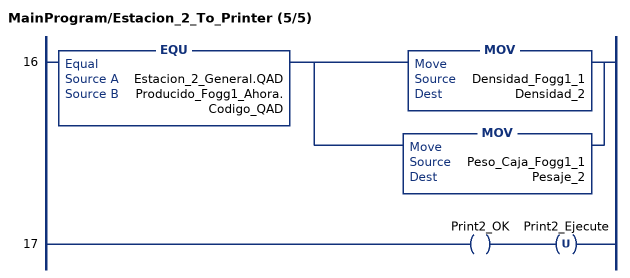
   16: EQU(Estacion_2_General.QAD,Producido_Fogg1_Ahora.Codigo_QAD)[MOV(Densidad_Fogg1_1,Densidad_2) ,MOV(Peso_Caja_Fogg1_1,Pesaje_2) ];
   17: OTE(Print2_OK)OTU(Print2_Ejecute);
END_ROUTINE
